# EPICS autosave request: support/ip-2-10/ipApp/Db/TSP_settings.req
#FILE... TSP_settings.req
#USAGE... TSP.db fields autosave'd.
$(P)$(TSP)TSP_FIL
$(P)$(TSP)TSP_AUTO_ADV
$(P)$(TSP)TSP_VALUE
$(P)$(TSP)TSP_UNITS
$(P)$(TSP)TSP_SECONDS
$(P)$(TSP)TSP_MINUTES
$(P)$(TSP)TSP_NCYCLES
$(P)$(TSP)TSP_MIN_PRESS
$(P)$(TSP)TSP_STAT.SCAN
